              Waypoint Linea28_B: TCP in base x=-638.706 y=351.254 z=110.848 mm, rx=0.1163 ry=3.1217 rz=0.0052 rad; joints [-32.94, -74.396, 108.519, -33.495, -217.835, -0.377] deg
              Folder bajada_comprobacion
                MoveDirectionNode (selectedDirection=ZMinus toolParams=0.1, 0.15)
                  Until DISTANCE (allowActions=false deceleration=3 distanceNodeType=STOP) Distance=0.071; motionParameters(blendRadius=0)
                MoveDirectionNode (selectedDirection=ZMinus toolParams=0.007, 0.007)
                  Until TOOL_CONTACT_DETECTION (allowActions=false retraction=0 decelerationAcceleration=0.02 decelerationAngularAcceleration=34.906585)
                MoveDirectionNode (selectedDirection=ZPlus toolParams=0.1, 0.15)
                  Until DISTANCE (allowActions=false deceleration=3 distanceNodeType=STOP) Distance=0.08; motionParameters(blendRadius=0)
          Folder AB
            'desbaste_inicial'
            bajada_broca := p[0,0,-0.008,0,0,0]
            barrenos_menos1 := 0
            barreno_actual := 0
            Loop While (checkContinuously=false) expression=barreno_actual≤barrenos_menos1
              Folder Perforacion
                MoveL speed 100 mm/s, acceleration 500 mm/s^2 (useActiveTCP=true) feature=Base
                  SuppressedNode
                    If barreno_actual≟3
                      barreno_actual := barreno_actual+1
                  SuppressedNode
                    internos := interpolate_pose(Linea28_B, Linea28_B, barreno_actual/barrenos_menos1)
                  SuppressedNode
                    Waypoint Waypoint (Variable): variable=internos
                  Waypoint Linea28_B referenceName=Linea28_B: TCP in base x=-638.706 y=351.254 z=110.848 mm, rx=0.1163 ry=3.1217 rz=0.0052 rad; joints [-32.94, -74.396, 108.519, -33.495, -217.835, -0.377] deg
                  'desbaste_inicial'
                  bajada_broca := p[0,0,-0.024,0,0,0]
                  bajada := p[0,0,0.024,0,0,0]
                  MoveDirectionNode (selectedDirection=ZMinus toolParams=0.1, 0.15)
                    Until DISTANCE (allowActions=false deceleration=3 distanceNodeType=STOP) Distance=0.071; motionParameters(blendRadius=0)
                  MoveDirectionNode (selectedDirection=ZMinus toolParams=0.007, 0.007)
                    Until TOOL_CONTACT_DETECTION (allowActions=false retraction=0 decelerationAcceleration=0.02 decelerationAngularAcceleration=34.906585)
                  Popup Message (haltProgram=false message=punto contacto alanzdo inputType=Text)
                  MoveDirectionNode (selectedDirection=ZPlus toolParams=0.015, 0.015)
                    Until DISTANCE (allowActions=false deceleration=3 distanceNodeType=STOP) Distance=0.01; motionParameters(blendRadius=0)
                  Wait Sleep waitTime=0.3
                  Set DigitalOutput pin=config_out[1]; digitalValue=1
                  Wait Sleep waitTime=0.3
                  Loop Counting (count=1) loopVariable(name=Loop_146)
                    bajar := pose_add(get_actual_tcp_pose(), bajada_broca)
                    Waypoint Waypoint (Variable): motionParameters(jointSpeed=1.047198 jointAcceleration=1.396263 cartesianSpeed=0.004 cartesianAcceleration=0.004); variable=bajar
                    subir := pose_sub(get_actual_tcp_pose(), bajada_broca)
                    MoveDirectionNode (selectedDirection=ZPlus toolParams=0.015, 0.015)
                      Until DISTANCE (allowActions=false deceleration=3 distanceNodeType=STOP) Distance=0.002; motionParameters(blendRadius=0)
                    Set DigitalOutput pin=config_out[1]; digitalValue=0
                    Waypoint Waypoint (Variable): motionParameters(jointSpeed=1.047198 jointAcceleration=1.396263 cartesianSpeed=0.015 cartesianAcceleration=0.015); variable=subir
                    bajada_broca := pose_sub(bajada_broca, bajada)
                  MoveDirectionNode (selectedDirection=ZPlus toolParams=0.1, 0.15)
                    Until DISTANCE (allowActions=false deceleration=3 distanceNodeType=STOP) Distance=0.08; motionParameters(blendRadius=0)
                  Set DigitalOutput pin=config_out[1]; digitalValue=0
                  barreno_actual := barreno_actual+1
                  SuppressedNode
                    Call Quitar_broca
                  SuppressedNode
                    Call Poner_broca
        Popup Message (haltProgram=false message=Linea28 con chica Terminada! inputType=Text)
        Folder Linea29
          Folder Marcar_puntos
            MoveL speed 100 mm/s, acceleration 500 mm/s^2 (useActiveTCP=true) feature=Base
              Waypoint Linea29_A: TCP in base x=-697.642 y=-428.593 z=109.99 mm, rx=-2.8017 ry=1.4172 rz=0.0072 rad; joints [13.48, -73.278, 107.072, -33.144, -302.021, -0.481] deg; TCP offset x=0.411 y=-218.298 z=37.994 mm, rx=1.558 ry=-0.1255 rz=0.1212 rad
              SuppressedNode
                Waypoint Linea29_BA: TCP in base x=-927.927 y=-428.7 z=110.397 mm, rx=-2.8034 ry=1.4179 rz=0.011 rad; joints [9.956, -55.686, 80.201, -24.007, -305.531, -0.529] deg
              Folder bajada_comprobacion
                MoveDirectionNode (selectedDirection=ZMinus toolParams=0.1, 0.15)
                  Until DISTANCE (allowActions=false deceleration=3 distanceNodeType=STOP) Distance=0.071; motionParameters(blendRadius=0)
                MoveDirectionNode (selectedDirection=ZMinus toolParams=0.007, 0.007)
                  Until TOOL_CONTACT_DETECTION (allowActions=false retraction=0 decelerationAcceleration=0.02 decelerationAngularAcceleration=34.906585)
                MoveDirectionNode (selectedDirection=ZPlus toolParams=0.1, 0.15)
                  Until DISTANCE (allowActions=false deceleration=3 distanceNodeType=STOP) Distance=0.08; motionParameters(blendRadius=0)
              SuppressedNode
                Waypoint Linea29_B: TCP in base x=-1160.231 y=-428.651 z=110.797 mm, rx=-2.8017 ry=1.4172 rz=0.0072 rad; joints [7.841, -31.782, 37.108, -4.619, -307.592, -0.568] deg
              Waypoint Linea29_AB: TCP in base x=-904.922 y=-428.637 z=110.457 mm, rx=-2.8017 ry=1.4172 rz=0.0072 rad; joints [10.222, -57.489, 83.131, -24.963, -305.263, -0.527] deg
              Folder bajada_comprobacion
                MoveDirectionNode (selectedDirection=ZMinus toolParams=0.1, 0.15)
                  Until DISTANCE (allowActions=false deceleration=3 distanceNodeType=STOP) Distance=0.071; motionParameters(blendRadius=0)
                MoveDirectionNode (selectedDirection=ZMinus toolParams=0.007, 0.007)
                  Until TOOL_CONTACT_DETECTION (allowActions=false retraction=0 decelerationAcceleration=0.02 decelerationAngularAcceleration=34.906585)
                MoveDirectionNode (selectedDirection=ZPlus toolParams=0.1, 0.15)
                  Until DISTANCE (allowActions=false deceleration=3 distanceNodeType=STOP) Distance=0.08; motionParameters(blendRadius=0)
          Folder AB
            'desbaste_inicial'
            bajada_broca := p[0,0,-0.008,0,0,0]
            barrenos_menos1 := 9
            barreno_actual := 0
            Loop While (checkContinuously=false) expression=barreno_actual≤barrenos_menos1
              Folder Perforacion
                MoveL speed 100 mm/s, acceleration 500 mm/s^2 (useActiveTCP=true) feature=Base
                  If barreno_actual≟7
                    barreno_actual := barreno_actual+1
                  internos := interpolate_pose(Linea29_A, Linea29_AB, barreno_actual/barrenos_menos1)
                  SuppressedNode
                    If barreno_actual≟6
                      MoveDirectionNode (selectedDirection=ZPlus)
                        Until DISTANCE (allowActions=false deceleration=3 distanceNodeType=STOP) Distance=0.01; motionParameters(blendRadius=0)
                  Waypoint Waypoint (Variable): variable=internos
                  'desbaste_inicial'
                  bajada_broca := p[0,0,-0.024,0,0,0]
                  bajada := p[0,0,0.024,0,0,0]
                  MoveDirectionNode (selectedDirection=ZMinus toolParams=0.1, 0.15)
                    Until DISTANCE (allowActions=false deceleration=3 distanceNodeType=STOP) Distance=0.071; motionParameters(blendRadius=0)
                  MoveDirectionNode (selectedDirection=ZMinus toolParams=0.007, 0.007)
                    Until TOOL_CONTACT_DETECTION (allowActions=false retraction=0 decelerationAcceleration=0.02 decelerationAngularAcceleration=34.906585)
                  Popup Message (haltProgram=false message=punto contacto alanzdo inputType=Text)
                  MoveDirectionNode (selectedDirection=ZPlus toolParams=0.015, 0.015)
                    Until DISTANCE (allowActions=false deceleration=3 distanceNodeType=STOP) Distance=0.007; motionParameters(blendRadius=0)
                  Wait Sleep waitTime=0.3
                  Set DigitalOutput pin=config_out[1]; digitalValue=1
                  Wait Sleep waitTime=0.3
                  Loop Counting (count=1) loopVariable(name=Loop_150)
                    bajar := pose_add(get_actual_tcp_pose(), bajada_broca)
                    Waypoint Waypoint (Variable): motionParameters(jointSpeed=1.047198 jointAcceleration=1.396263 cartesianSpeed=0.004 cartesianAcceleration=0.004); variable=bajar
                    subir := pose_sub(get_actual_tcp_pose(), bajada_broca)
                    MoveDirectionNode (selectedDirection=ZPlus toolParams=0.015, 0.015)
                      Until DISTANCE (allowActions=false deceleration=3 distanceNodeType=STOP) Distance=0.002; motionParameters(blendRadius=0)
                    Set DigitalOutput pin=config_out[1]; digitalValue=0
                    Waypoint Waypoint (Variable): motionParameters(jointSpeed=1.047198 jointAcceleration=1.396263 cartesianSpeed=0.015 cartesianAcceleration=0.015); variable=subir
                    bajada_broca := pose_sub(bajada_broca, bajada)
                  MoveDirectionNode (selectedDirection=ZPlus toolParams=0.1, 0.15)
                    Until DISTANCE (allowActions=false deceleration=3 distanceNodeType=STOP) Distance=0.04; motionParameters(blendRadius=0)
                  Set DigitalOutput pin=config_out[1]; digitalValue=0
                  barreno_actual := barreno_actual+1
                  SuppressedNode
                    Call Quitar_broca
                  SuppressedNode
                    Call Poner_broca
        Folder Linea29B
          Folder Marcar_puntos
            MoveL speed 100 mm/s, acceleration 500 mm/s^2 (useActiveTCP=true) feature=Base
              SuppressedNode
                Waypoint Linea29_A: TCP in base x=-697.642 y=-428.593 z=109.99 mm, rx=-2.8017 ry=1.4172 rz=0.0072 rad; joints [13.48, -73.278, 107.072, -33.144, -302.021, -0.481] deg
              Waypoint Linea29_BA: TCP in base x=-927.927 y=-428.7 z=110.397 mm, rx=-2.8034 ry=1.4179 rz=0.011 rad; joints [9.956, -55.686, 80.201, -24.007, -305.531, -0.529] deg
              Folder bajada_comprobacion
                MoveDirectionNode (selectedDirection=ZMinus toolParams=0.1, 0.15)
                  Until DISTANCE (allowActions=false deceleration=3 distanceNodeType=STOP) Distance=0.071; motionParameters(blendRadius=0)
                MoveDirectionNode (selectedDirection=ZMinus toolParams=0.007, 0.007)
                  Until TOOL_CONTACT_DETECTION (allowActions=false retraction=0 decelerationAcceleration=0.02 decelerationAngularAcceleration=34.906585)
                MoveDirectionNode (selectedDirection=ZPlus toolParams=0.1, 0.15)
                  Until DISTANCE (allowActions=false deceleration=3 distanceNodeType=STOP) Distance=0.08; motionParameters(blendRadius=0)
              Waypoint Linea29_B: TCP in base x=-1160.231 y=-428.651 z=110.797 mm, rx=-2.8017 ry=1.4172 rz=0.0072 rad; joints [7.841, -31.782, 37.108, -4.619, -307.592, -0.568] deg
              SuppressedNode
                Waypoint Linea29_AB: TCP in base x=-904.922 y=-428.637 z=110.457 mm, rx=-2.8017 ry=1.4172 rz=0.0072 rad; joints [10.222, -57.489, 83.131, -24.963, -305.263, -0.527] deg
              Folder bajada_comprobacion
                MoveDirectionNode (selectedDirection=ZMinus toolParams=0.1, 0.15)
                  Until DISTANCE (allowActions=false deceleration=3 distanceNodeType=STOP) Distance=0.071; motionParameters(blendRadius=0)
                MoveDirectionNode (selectedDirection=ZMinus toolParams=0.007, 0.007)
                  Until TOOL_CONTACT_DETECTION (allowActions=false retraction=0 decelerationAcceleration=0.02 decelerationAngularAcceleration=34.906585)
                MoveDirectionNode (selectedDirection=ZPlus toolParams=0.1, 0.15)
                  Until DISTANCE (allowActions=false deceleration=3 distanceNodeType=STOP) Distance=0.08; motionParameters(blendRadius=0)
          Folder AB
            'desbaste_inicial'
            bajada_broca := p[0,0,-0.008,0,0,0]
            barrenos_menos1 := 10
            barreno_actual := 5
            Loop While (checkContinuously=false) expression=barreno_actual≤barrenos_menos1
              Folder Perforacion
                MoveL speed 100 mm/s, acceleration 500 mm/s^2 (useActiveTCP=true) feature=Base
                  SuppressedNode
                    If barreno_actual≟7
                      barreno_actual := barreno_actual+1
                  internos := interpolate_pose(Linea29_BA, Linea29_B, barreno_actual/barrenos_menos1)
                  SuppressedNode
                    If barreno_actual≟6
                      MoveDirectionNode (selectedDirection=ZPlus)
                        Until DISTANCE (allowActions=false deceleration=3 distanceNodeType=STOP) Distance=0.01; motionParameters(blendRadius=0)
                  Waypoint Waypoint (Variable): variable=internos
                  'desbaste_inicial'
                  bajada_broca := p[0,0,-0.024,0,0,0]
                  bajada := p[0,0,0.024,0,0,0]
                  MoveDirectionNode (selectedDirection=ZMinus toolParams=0.1, 0.15)
                    Until DISTANCE (allowActions=false deceleration=3 distanceNodeType=STOP) Distance=0.071; motionParameters(blendRadius=0)
                  MoveDirectionNode (selectedDirection=ZMinus toolParams=0.007, 0.007)
                    Until TOOL_CONTACT_DETECTION (allowActions=false retraction=0 decelerationAcceleration=0.02 decelerationAngularAcceleration=34.906585)
                  Popup Message (haltProgram=false message=punto contacto alanzdo inputType=Text)
                  MoveDirectionNode (selectedDirection=ZPlus toolParams=0.015, 0.015)
                    Until DISTANCE (allowActions=false deceleration=3 distanceNodeType=STOP) Distance=0.007; motionParameters(blendRadius=0)
                  Wait Sleep waitTime=0.3
                  Set DigitalOutput pin=config_out[1]; digitalValue=1
                  Wait Sleep waitTime=0.3
                  Loop Counting (count=1) loopVariable(name=Loop_30)
                    bajar := pose_add(get_actual_tcp_pose(), bajada_broca)
                    Waypoint Waypoint (Variable): motionParameters(jointSpeed=1.047198 jointAcceleration=1.396263 cartesianSpeed=0.004 cartesianAcceleration=0.004); variable=bajar
                    subir := pose_sub(get_actual_tcp_pose(), bajada_broca)
                    MoveDirectionNode (selectedDirection=ZPlus toolParams=0.015, 0.015)
                      Until DISTANCE (allowActions=false deceleration=3 distanceNodeType=STOP) Distance=0.002; motionParameters(blendRadius=0)
                    Set DigitalOutput pin=config_out[1]; digitalValue=0
                    Waypoint Waypoint (Variable): motionParameters(jointSpeed=1.047198 jointAcceleration=1.396263 cartesianSpeed=0.015 cartesianAcceleration=0.015); variable=subir
                    bajada_broca := pose_sub(bajada_broca, bajada)
                  MoveDirectionNode (selectedDirection=ZPlus toolParams=0.1, 0.15)
                    Until DISTANCE (allowActions=false deceleration=3 distanceNodeType=STOP) Distance=0.04; motionParameters(blendRadius=0)
                  Set DigitalOutput pin=config_out[1]; digitalValue=0
                  barreno_actual := barreno_actual+1
                  SuppressedNode
                    Call Quitar_broca
                  SuppressedNode
                    Call Poner_broca
        Popup Message (haltProgram=false message=Linea29 con chica Terminada! inputType=Text)
      SuppressedNode
        Folder Broca_2
          Folder Linea7
            Folder Marcar_puntos
              MoveL speed 100 mm/s, acceleration 500 mm/s^2 (useActiveTCP=true) feature=Base
                Waypoint Home2: TCP in base x=-476.229 y=0 z=568.737 mm, rx=2.0263 ry=-2.3929 rz=-0.0208 rad; joints [-32.551, -116.469, 98.413, 17.843, -302.102, -0.163] deg; TCP offset x=0.411 y=-218.298 z=37.994 mm, rx=1.558 ry=-0.1255 rz=0.1212 rad
                Waypoint Linea7_A: TCP in base x=-749.561 y=-351.839 z=110.843 mm, rx=3.1084 ry=-0.3759 rz=-0.0174 rad; joints [1.917, -65.95, 96.598, -30.808, -353.455, -0.309] deg
                Waypoint Linea7_B: TCP in base x=-795.37 y=-351.638 z=110.748 mm, rx=3.1084 ry=-0.3758 rz=-0.0174 rad; joints [1.792, -62.243, 90.906, -28.822, -353.578, -0.309] deg
            Folder AB
              'desbaste_inicial'
              bajada_broca := p[0,0,-0.008,0,0,0]
              barrenos_menos1 := 2
              barreno_actual := 0
              Loop While (checkContinuously=false) expression=barreno_actual≤barrenos_menos1
                Folder Perforacion
                  MoveL speed 100 mm/s, acceleration 500 mm/s^2 (useActiveTCP=true) feature=Base
                    internos := interpolate_pose(Linea7_A, Linea7_B, barreno_actual/barrenos_menos1)
                    Waypoint Waypoint (Variable): variable=internos
                    'desbaste_inicial'
                    bajada_broca := p[0,0,-0.008,0,0,0]
                    bajada := p[0,0,0.008,0,0,0]
                    MoveDirectionNode (selectedDirection=ZMinus toolParams=0.003, 0.005)
                      Until DISTANCE (allowActions=false deceleration=3 distanceNodeType=STOP) Distance=0.045; motionParameters(blendRadius=0)
                    Popup Message (haltProgram=false message=punto contacto alanzdo inputType=Text)
                    MoveDirectionNode (selectedDirection=ZPlus toolParams=0.003, 0.005)
                      Until DISTANCE (allowActions=false deceleration=3 distanceNodeType=STOP) Distance=0.002; motionParameters(blendRadius=0)
                    Wait Sleep waitTime=0.3
                    Set DigitalOutput pin=config_out[1]; digitalValue=1
                    Wait Sleep waitTime=0.3
                    Loop Counting (count=3) loopVariable(name=Loop_111)
                      bajar := pose_add(get_actual_tcp_pose(), bajada_broca)
                      Waypoint Waypoint (Variable): motionParameters(jointSpeed=1.047198 jointAcceleration=1.396263 cartesianSpeed=0.001 cartesianAcceleration=0.005); variable=bajar
                      subir := pose_sub(get_actual_tcp_pose(), bajada_broca)
                      Waypoint Waypoint (Variable): motionParameters(jointSpeed=1.047198 jointAcceleration=1.396263 cartesianSpeed=0.005 cartesianAcceleration=0.01); variable=subir
                      bajada_broca := pose_sub(bajada_broca, bajada)
                    MoveDirectionNode (selectedDirection=ZPlus toolParams=0.03, 0.035)
                      Until DISTANCE (allowActions=false deceleration=3 distanceNodeType=STOP) Distance=0.06; motionParameters(blendRadius=0)
                    Set DigitalOutput pin=config_out[1]; digitalValue=0
                    barreno_actual := barreno_actual+1
                    SuppressedNode
                      Call Quitar_broca
                    SuppressedNode
                      Call Poner_broca
          Popup Message (haltProgram=false message=Linea7 con chica Terminada! inputType=Text)
          Folder Linea8
            Folder Marcar_puntos
              MoveL speed 100 mm/s, acceleration 500 mm/s^2 (useActiveTCP=true) feature=Base
                Waypoint Linea8_A: TCP in base x=-897.665 y=-351.421 z=100.251 mm, rx=3.1084 ry=-0.3758 rz=-0.0174 rad; joints [1.574, -53.233, 77.321, -24.256, -353.784, -0.302] deg
                Waypoint Linea8_B: TCP in base x=-1021.743 y=-350.913 z=110.77 mm, rx=3.1084 ry=-0.3758 rz=-0.0173 rad; joints [1.351, -41.656, 55.75, -14.225, -353.984, -0.335] deg
            Folder AB
              'desbaste_inicial'
              bajada_broca := p[0,0,-0.008,0,0,0]
              barrenos_menos1 := 5
              barreno_actual := 0
              Loop While (checkContinuously=false) expression=barreno_actual≤barrenos_menos1
                Folder Perforacion
                  MoveL speed 100 mm/s, acceleration 500 mm/s^2 (useActiveTCP=true) feature=Base
                    internos := interpolate_pose(Linea8_A, Linea8_B, barreno_actual/barrenos_menos1)
                    Waypoint Waypoint (Variable): variable=internos
                    'desbaste_inicial'
                    bajada_broca := p[0,0,-0.008,0,0,0]
                    bajada := p[0,0,0.008,0,0,0]
                    MoveDirectionNode (selectedDirection=ZMinus toolParams=0.003, 0.005)
                      Until DISTANCE (allowActions=false deceleration=3 distanceNodeType=STOP) Distance=0.045; motionParameters(blendRadius=0)
                    Popup Message (haltProgram=false message=punto contacto alanzdo inputType=Text)
                    MoveDirectionNode (selectedDirection=ZPlus toolParams=0.003, 0.005)
                      Until DISTANCE (allowActions=false deceleration=3 distanceNodeType=STOP) Distance=0.002; motionParameters(blendRadius=0)
                    Wait Sleep waitTime=0.3
                    Set DigitalOutput pin=config_out[1]; digitalValue=1
                    Wait Sleep waitTime=0.3
                    Loop Counting (count=3) loopVariable(name=Loop_113)
                      bajar := pose_add(get_actual_tcp_pose(), bajada_broca)
                      Waypoint Waypoint (Variable): motionParameters(jointSpeed=1.047198 jointAcceleration=1.396263 cartesianSpeed=0.001 cartesianAcceleration=0.005); variable=bajar
                      subir := pose_sub(get_actual_tcp_pose(), bajada_broca)
                      Waypoint Waypoint (Variable): motionParameters(jointSpeed=1.047198 jointAcceleration=1.396263 cartesianSpeed=0.005 cartesianAcceleration=0.01); variable=subir
                      bajada_broca := pose_sub(bajada_broca, bajada)
                    MoveDirectionNode (selectedDirection=ZPlus toolParams=0.03, 0.035)
                      Until DISTANCE (allowActions=false deceleration=3 distanceNodeType=STOP) Distance=0.06; motionParameters(blendRadius=0)
                    Set DigitalOutput pin=config_out[1]; digitalValue=0
                    barreno_actual := barreno_actual+1
                    SuppressedNode
                      Call Quitar_broca
                    SuppressedNode
                      Call Poner_broca
          Popup Message (haltProgram=false message=Linea8 con chica Terminada! inputType=Text)
          Folder Linea9
            Folder Marcar_puntos
              MoveL speed 100 mm/s, acceleration 500 mm/s^2 (useActiveTCP=true) feature=Base
                Waypoint Linea9_A: TCP in base x=-1101.087 y=-350.536 z=110.686 mm, rx=3.1084 ry=-0.3759 rz=-0.0174 rad; joints [1.23, -31.558, 36.849, -5.411, -354.078, -0.351] deg
                Waypoint Linea9_B: TCP in base x=-1151 y=-350.505 z=110.708 mm, rx=3.1084 ry=-0.3759 rz=-0.0174 rad; joints [1.169, -21.153, 16.449, 4.577, -354.109, -0.341] deg
            Folder AB
              'desbaste_inicial'
              bajada_broca := p[0,0,-0.008,0,0,0]
              barrenos_menos1 := 2
              barreno_actual := 0
              Loop While (checkContinuously=false) expression=barreno_actual≤barrenos_menos1
                Folder Perforacion
                  MoveL speed 100 mm/s, acceleration 500 mm/s^2 (useActiveTCP=true) feature=Base
                    internos := interpolate_pose(Linea9_A, Linea9_B, barreno_actual/barrenos_menos1)
                    Waypoint Waypoint (Variable): variable=internos
                    'desbaste_inicial'
                    bajada_broca := p[0,0,-0.008,0,0,0]
                    bajada := p[0,0,0.008,0,0,0]
                    MoveDirectionNode (selectedDirection=ZMinus toolParams=0.003, 0.005)
                      Until DISTANCE (allowActions=false deceleration=3 distanceNodeType=STOP) Distance=0.045; motionParameters(blendRadius=0)
                    Popup Message (haltProgram=false message=punto contacto alanzdo inputType=Text)
                    MoveDirectionNode (selectedDirection=ZPlus toolParams=0.003, 0.005)
                      Until DISTANCE (allowActions=false deceleration=3 distanceNodeType=STOP) Distance=0.002; motionParameters(blendRadius=0)
                    Wait Sleep waitTime=0.3
                    Set DigitalOutput pin=config_out[1]; digitalValue=1
                    Wait Sleep waitTime=0.3
                    Loop Counting (count=3) loopVariable(name=Loop_115)
                      bajar := pose_add(get_actual_tcp_pose(), bajada_broca)
                      Waypoint Waypoint (Variable): motionParameters(jointSpeed=1.047198 jointAcceleration=1.396263 cartesianSpeed=0.001 cartesianAcceleration=0.005); variable=bajar
                      subir := pose_sub(get_actual_tcp_pose(), bajada_broca)
                      Waypoint Waypoint (Variable): motionParameters(jointSpeed=1.047198 jointAcceleration=1.396263 cartesianSpeed=0.005 cartesianAcceleration=0.01); variable=subir
                      bajada_broca := pose_sub(bajada_broca, bajada)
                    MoveDirectionNode (selectedDirection=ZPlus toolParams=0.03, 0.035)
                      Until DISTANCE (allowActions=false deceleration=3 distanceNodeType=STOP) Distance=0.06; motionParameters(blendRadius=0)
                    Set DigitalOutput pin=config_out[1]; digitalValue=0
                    barreno_actual := barreno_actual+1
                    SuppressedNode
                      Call Quitar_broca
                    SuppressedNode
                      Call Poner_broca
          Popup Message (haltProgram=false message=Linea9 con chica Terminada! inputType=Text)
          Folder Linea10
            Folder Marcar_puntos
              MoveL speed 100 mm/s, acceleration 500 mm/s^2 (useActiveTCP=true) feature=Base
                Waypoint Home2: TCP in base x=-476.229 y=0 z=568.737 mm, rx=2.0263 ry=-2.3929 rz=-0.0208 rad; joints [-32.551, -116.469, 98.413, 17.843, -302.102, -0.163] deg
                Waypoint Linea10_A: TCP in base x=-634.372 y=-317.237 z=110 mm, rx=3.1084 ry=-0.3759 rz=-0.0173 rad; joints [-0.923, -75.994, 110.915, -35.183, -356.299, -0.201] deg
                Waypoint Linea10_B: TCP in base x=-637.528 y=-266.765 z=110 mm, rx=2.0205 ry=-2.3939 rz=-0.0206 rad; joints [10.666, -83.833, 120.67, -37.235, -258.835, -0.176] deg
            Folder AB
              'desbaste_inicial'
              bajada_broca := p[0,0,-0.008,0,0,0]
              barrenos_menos1 := 2
              barreno_actual := 0
              Loop While (checkContinuously=false) expression=barreno_actual≤barrenos_menos1
                Folder Perforacion
                  MoveL speed 100 mm/s, acceleration 500 mm/s^2 (useActiveTCP=true) feature=Base
                    internos := interpolate_pose(Linea10_A, Linea10_B, barreno_actual/barrenos_menos1)
                    Waypoint Waypoint (Variable): variable=internos
                    'desbaste_inicial'
                    bajada_broca := p[0,0,-0.008,0,0,0]
                    bajada := p[0,0,0.008,0,0,0]
                    MoveDirectionNode (selectedDirection=ZMinus toolParams=0.003, 0.005)
                      Until DISTANCE (allowActions=false deceleration=3 distanceNodeType=STOP) Distance=0.045; motionParameters(blendRadius=0)
                    Popup Message (haltProgram=false message=punto contacto alanzdo inputType=Text)
                    MoveDirectionNode (selectedDirection=ZPlus toolParams=0.003, 0.005)
                      Until DISTANCE (allowActions=false deceleration=3 distanceNodeType=STOP) Distance=0.002; motionParameters(blendRadius=0)
                    Wait Sleep waitTime=0.3
                    Set DigitalOutput pin=config_out[1]; digitalValue=1
                    Wait Sleep waitTime=0.3
                    Loop Counting (count=3) loopVariable(name=Loop_117)
                      bajar := pose_add(get_actual_tcp_pose(), bajada_broca)
                      Waypoint Waypoint (Variable): motionParameters(jointSpeed=1.047198 jointAcceleration=1.396263 cartesianSpeed=0.001 cartesianAcceleration=0.005); variable=bajar
                      subir := pose_sub(get_actual_tcp_pose(), bajada_broca)
                      Waypoint Waypoint (Variable): motionParameters(jointSpeed=1.047198 jointAcceleration=1.396263 cartesianSpeed=0.005 cartesianAcceleration=0.01); variable=subir
                      bajada_broca := pose_sub(bajada_broca, bajada)
                    MoveDirectionNode (selectedDirection=ZPlus toolParams=0.03, 0.035)
                      Until DISTANCE (allowActions=false deceleration=3 distanceNodeType=STOP) Distance=0.06; motionParameters(blendRadius=0)
                    Set DigitalOutput pin=config_out[1]; digitalValue=0
                    barreno_actual := barreno_actual+1
                    SuppressedNode
                      Call Quitar_broca
                    SuppressedNode
                      Call Poner_broca
          Popup Message (haltProgram=false message=Linea10 con chica Terminada! inputType=Text)
          Folder Linea11
            Folder Marcar_puntos
              MoveL speed 100 mm/s, acceleration 500 mm/s^2 (useActiveTCP=true) feature=Base
                Waypoint Linea11_A: TCP in base x=-636.9 y=-137.433 z=110 mm, rx=2.0204 ry=-2.394 rz=-0.0205 rad; joints [-4.253, -88.617, 125.878, -37.636, -273.75, -0.078] deg
                Waypoint Linea11_B: TCP in base x=-636.767 y=-82.891 z=110 mm, rx=2.0204 ry=-2.3939 rz=-0.0206 rad; joints [-10.939, -89.848, 127.132, -37.66, -280.436, -0.033] deg
            Folder AB
              'desbaste_inicial'
              bajada_broca := p[0,0,-0.008,0,0,0]
              barrenos_menos1 := 2
              barreno_actual := 0
              Loop While (checkContinuously=false) expression=barreno_actual≤barrenos_menos1
                Folder Perforacion
                  MoveL speed 100 mm/s, acceleration 500 mm/s^2 (useActiveTCP=true) feature=Base
                    SuppressedNode
                      If barreno_actual≟5
                        barreno_actual := barreno_actual+1
                    internos := interpolate_pose(Linea11_A, Linea11_B, barreno_actual/barrenos_menos1)
                    Waypoint Waypoint (Variable): variable=internos
                    'desbaste_inicial'
                    bajada_broca := p[0,0,-0.008,0,0,0]
                    bajada := p[0,0,0.008,0,0,0]
                    MoveDirectionNode (selectedDirection=ZMinus toolParams=0.003, 0.005)
                      Until DISTANCE (allowActions=false deceleration=3 distanceNodeType=STOP) Distance=0.045; motionParameters(blendRadius=0)
                    Popup Message (haltProgram=false message=punto contacto alanzdo inputType=Text)
                    MoveDirectionNode (selectedDirection=ZPlus toolParams=0.003, 0.005)
                      Until DISTANCE (allowActions=false deceleration=3 distanceNodeType=STOP) Distance=0.002; motionParameters(blendRadius=0)
                    Wait Sleep waitTime=0.3
                    Set DigitalOutput pin=config_out[1]; digitalValue=1
                    Wait Sleep waitTime=0.3
                    Loop Counting (count=3) loopVariable(name=Loop_119)
                      bajar := pose_add(get_actual_tcp_pose(), bajada_broca)
                      Waypoint Waypoint (Variable): motionParameters(jointSpeed=1.047198 jointAcceleration=1.396263 cartesianSpeed=0.001 cartesianAcceleration=0.005); variable=bajar
                      subir := pose_sub(get_actual_tcp_pose(), bajada_broca)
                      Waypoint Waypoint (Variable): motionParameters(jointSpeed=1.047198 jointAcceleration=1.396263 cartesianSpeed=0.005 cartesianAcceleration=0.01); variable=subir
                      bajada_broca := pose_sub(bajada_broca, bajada)
                    MoveDirectionNode (selectedDirection=ZPlus toolParams=0.03, 0.035)
                      Until DISTANCE (allowActions=false deceleration=3 distanceNodeType=STOP) Distance=0.06; motionParameters(blendRadius=0)
                    Set DigitalOutput pin=config_out[1]; digitalValue=0
                    barreno_actual := barreno_actual+1
                    SuppressedNode
                      Call Quitar_broca
                    SuppressedNode
                      Call Poner_broca
          Popup Message (haltProgram=false message=Linea11 con chica Terminada! inputType=Text)
          Folder Linea12
            Folder Marcar_puntos
              MoveL speed 100 mm/s, acceleration 500 mm/s^2 (useActiveTCP=true) feature=Base
                Waypoint Linea12_A: TCP in base x=-636.731 y=-59.028 z=110 mm, rx=2.0204 ry=-2.3939 rz=-0.0205 rad; joints [-13.873, -90.206, 127.489, -37.657, -283.371, -0.016] deg
                Waypoint Linea12_B: TCP in base x=-636.063 y=114.709 z=110 mm, rx=2.0204 ry=-2.3939 rz=-0.0206 rad; joints [-33.88, -89.351, 126.631, -37.694, -303.38, 0.135] deg
            Folder AB
              'desbaste_inicial'
              bajada_broca := p[0,0,-0.008,0,0,0]
              barrenos_menos1 := 7
              barreno_actual := 0
              Loop While (checkContinuously=false) expression=barreno_actual≤barrenos_menos1
                Folder Perforacion
                  MoveL speed 100 mm/s, acceleration 500 mm/s^2 (useActiveTCP=true) feature=Base
                    If barreno_actual≟2
                      barreno_actual := barreno_actual+1
                    internos := interpolate_pose(Linea12_A, Linea12_B, barreno_actual/barrenos_menos1)
                    Waypoint Waypoint (Variable): variable=internos
                    'desbaste_inicial'
                    bajada_broca := p[0,0,-0.008,0,0,0]
                    bajada := p[0,0,0.008,0,0,0]
                    MoveDirectionNode (selectedDirection=ZMinus toolParams=0.003, 0.005)
                      Until DISTANCE (allowActions=false deceleration=3 distanceNodeType=STOP) Distance=0.045; motionParameters(blendRadius=0)
                    Popup Message (haltProgram=false message=punto contacto alanzdo inputType=Text)
                    MoveDirectionNode (selectedDirection=ZPlus toolParams=0.003, 0.005)
                      Until DISTANCE (allowActions=false deceleration=3 distanceNodeType=STOP) Distance=0.002; motionParameters(blendRadius=0)
                    Wait Sleep waitTime=0.3
                    Set DigitalOutput pin=config_out[1]; digitalValue=1
                    Wait Sleep waitTime=0.3
                    Loop Counting (count=3) loopVariable(name=Loop_121)
                      bajar := pose_add(get_actual_tcp_pose(), bajada_broca)
                      Waypoint Waypoint (Variable): motionParameters(jointSpeed=1.047198 jointAcceleration=1.396263 cartesianSpeed=0.001 cartesianAcceleration=0.005); variable=bajar
                      subir := pose_sub(get_actual_tcp_pose(), bajada_broca)
                      Waypoint Waypoint (Variable): motionParameters(jointSpeed=1.047198 jointAcceleration=1.396263 cartesianSpeed=0.005 cartesianAcceleration=0.01); variable=subir
                      bajada_broca := pose_sub(bajada_broca, bajada)
                    MoveDirectionNode (selectedDirection=ZPlus toolParams=0.03, 0.035)
                      Until DISTANCE (allowActions=false deceleration=3 distanceNodeType=STOP) Distance=0.06; motionParameters(blendRadius=0)
                    Set DigitalOutput pin=config_out[1]; digitalValue=0
                    barreno_actual := barreno_actual+1
                    SuppressedNode
                      Call Quitar_broca
                    SuppressedNode
                      Call Poner_broca
          Popup Message (haltProgram=false message=Linea12 con chica Terminada! inputType=Text)
          Folder Linea13
            Folder Marcar_puntos
              MoveL speed 100 mm/s, acceleration 500 mm/s^2 (useActiveTCP=true) feature=Base
                Waypoint Linea13_A: TCP in base x=-636.036 y=270.318 z=110 mm, rx=2.0205 ry=-2.3939 rz=-0.0206 rad; joints [-47.614, -83.952, 120.807, -37.347, -317.114, 0.279] deg
                Waypoint Linea13_B: TCP in base x=-635.536 y=326.664 z=110 mm, rx=2.0205 ry=-2.3939 rz=-0.0206 rad; joints [-51.543, -81.32, 117.724, -36.932, -321.042, 0.336] deg
            Folder AB
              'desbaste_inicial'
              bajada_broca := p[0,0,-0.008,0,0,0]
              barrenos_menos1 := 2
              barreno_actual := 0
              Loop While (checkContinuously=false) expression=barreno_actual≤barrenos_menos1
                Folder Perforacion
                  MoveL speed 100 mm/s, acceleration 500 mm/s^2 (useActiveTCP=true) feature=Base
                    SuppressedNode
                      If barreno_actual≟2
                        barreno_actual := barreno_actual+1
                    internos := interpolate_pose(Linea13_A, Linea13_B, barreno_actual/barrenos_menos1)
                    Waypoint Waypoint (Variable): variable=internos
                    'desbaste_inicial'
                    bajada_broca := p[0,0,-0.008,0,0,0]
                    bajada := p[0,0,0.008,0,0,0]
                    MoveDirectionNode (selectedDirection=ZMinus toolParams=0.003, 0.005)
                      Until DISTANCE (allowActions=false deceleration=3 distanceNodeType=STOP) Distance=0.045; motionParameters(blendRadius=0)
                    Popup Message (haltProgram=false message=punto contacto alanzdo inputType=Text)
                    MoveDirectionNode (selectedDirection=ZPlus toolParams=0.003, 0.005)
                      Until DISTANCE (allowActions=false deceleration=3 distanceNodeType=STOP) Distance=0.002; motionParameters(blendRadius=0)
                    Wait Sleep waitTime=0.3
                    Set DigitalOutput pin=config_out[1]; digitalValue=1
                    Wait Sleep waitTime=0.3
                    Loop Counting (count=3) loopVariable=Loop_123
                      bajar := pose_add(get_actual_tcp_pose(), bajada_broca)
                      Waypoint Waypoint (Variable): motionParameters(jointSpeed=1.047198 jointAcceleration=1.396263 cartesianSpeed=0.001 cartesianAcceleration=0.005); variable=bajar
                      subir := pose_sub(get_actual_tcp_pose(), bajada_broca)
                      Waypoint Waypoint (Variable): motionParameters(jointSpeed=1.047198 jointAcceleration=1.396263 cartesianSpeed=0.005 cartesianAcceleration=0.01); variable=subir
                      bajada_broca := pose_sub(bajada_broca, bajada)
                    MoveDirectionNode (selectedDirection=ZPlus toolParams=0.03, 0.035)
                      Until DISTANCE (allowActions=false deceleration=3 distanceNodeType=STOP) Distance=0.06; motionParameters(blendRadius=0)
                    Set DigitalOutput pin=config_out[1]; digitalValue=0
                    barreno_actual := barreno_actual+1
                    SuppressedNode
                      Call Quitar_broca
                    SuppressedNode
                      Call Poner_broca
          Popup Message (haltProgram=false message=Linea13 con chica Terminada! inputType=Text)
          Folder Linea14
            Folder Marcar_puntos
              MoveL speed 100 mm/s, acceleration 500 mm/s^2 (useActiveTCP=true) feature=Base
                Waypoint Linea14_A: TCP in base x=-635.47 y=349.602 z=110 mm, rx=2.0205 ry=-2.3938 rz=-0.0205 rad; joints [-52.983, -80.161, 116.316, -36.699, -322.484, 0.362] deg
                Waypoint Linea14_B: TCP in base x=-634.908 y=491.921 z=110 mm, rx=2.0205 ry=-2.3939 rz=-0.0205 rad; joints [-60.308, -72.235, 105.919, -34.338, -329.805, 0.501] deg
            Folder AB
              'desbaste_inicial'
              bajada_broca := p[0,0,-0.008,0,0,0]
              barrenos_menos1 := 5
              barreno_actual := 0
              Loop While (checkContinuously=false) expression=barreno_actual≤barrenos_menos1
                Folder Perforacion
                  MoveL speed 100 mm/s, acceleration 500 mm/s^2 (useActiveTCP=true) feature=Base
                    If barreno_actual≟3
                      barreno_actual := barreno_actual+1
                    internos := interpolate_pose(Linea14_A, Linea14_B, barreno_actual/barrenos_menos1)
                    Waypoint Waypoint (Variable): variable=internos
                    'desbaste_inicial'
                    bajada_broca := p[0,0,-0.008,0,0,0]
                    bajada := p[0,0,0.008,0,0,0]
                    MoveDirectionNode (selectedDirection=ZMinus toolParams=0.003, 0.005)
                      Until DISTANCE (allowActions=false deceleration=3 distanceNodeType=STOP) Distance=0.045; motionParameters(blendRadius=0)
                    Popup Message (haltProgram=false message=punto contacto alanzdo inputType=Text)
                    MoveDirectionNode (selectedDirection=ZPlus toolParams=0.003, 0.005)
                      Until DISTANCE (allowActions=false deceleration=3 distanceNodeType=STOP) Distance=0.002; motionParameters(blendRadius=0)
                    Wait Sleep waitTime=0.3
                    Set DigitalOutput pin=config_out[1]; digitalValue=1
                    Wait Sleep waitTime=0.3
                    Loop Counting (count=3) loopVariable=Loop_125
                      bajar := pose_add(get_actual_tcp_pose(), bajada_broca)
                      Waypoint Waypoint (Variable): motionParameters(jointSpeed=1.047198 jointAcceleration=1.396263 cartesianSpeed=0.001 cartesianAcceleration=0.005); variable=bajar
                      subir := pose_sub(get_actual_tcp_pose(), bajada_broca)
                      Waypoint Waypoint (Variable): motionParameters(jointSpeed=1.047198 jointAcceleration=1.396263 cartesianSpeed=0.005 cartesianAcceleration=0.01); variable=subir
                      bajada_broca := pose_sub(bajada_broca, bajada)
                    MoveDirectionNode (selectedDirection=ZPlus toolParams=0.03, 0.035)
                      Until DISTANCE (allowActions=false deceleration=3 distanceNodeType=STOP) Distance=0.06; motionParameters(blendRadius=0)
                    Set DigitalOutput pin=config_out[1]; digitalValue=0
                    barreno_actual := barreno_actual+1
                    SuppressedNode
                      Call Quitar_broca
                    SuppressedNode
                      Call Poner_broca
          Popup Message (haltProgram=false message=Linea14 con chica Terminada! inputType=Text)
          Folder Linea15
            Folder Marcar_puntos
              MoveL speed 100 mm/s, acceleration 500 mm/s^2 (useActiveTCP=true) feature=Base
                Waypoint Linea15_A: TCP in base x=-634.597 y=515.429 z=110 mm, rx=2.0204 ry=-2.394 rz=-0.0205 rad; joints [-61.306, -70.837, 103.953, -33.788, -330.797, 0.523] deg
                Waypoint Linea15_B: TCP in base x=-634.619 y=593.839 z=110 mm, rx=2.0204 ry=-2.3939 rz=-0.0206 rad; joints [-64.194, -65.927, 96.758, -31.573, -333.685, 0.603] deg
            Folder AB
              'desbaste_inicial'
              bajada_broca := p[0,0,-0.008,0,0,0]
              barrenos_menos1 := 3
              barreno_actual := 0
              Loop While (checkContinuously=false) expression=barreno_actual≤barrenos_menos1
                Folder Perforacion
                  MoveL speed 100 mm/s, acceleration 500 mm/s^2 (useActiveTCP=true) feature=Base
                    SuppressedNode
                      If barreno_actual≟3
                        barreno_actual := barreno_actual+1
                    internos := interpolate_pose(Linea15_A, Linea15_B, barreno_actual/barrenos_menos1)
                    Waypoint Waypoint (Variable): variable=internos
                    'desbaste_inicial'
                    bajada_broca := p[0,0,-0.008,0,0,0]
                    bajada := p[0,0,0.008,0,0,0]
                    MoveDirectionNode (selectedDirection=ZMinus toolParams=0.003, 0.005)
                      Until DISTANCE (allowActions=false deceleration=3 distanceNodeType=STOP) Distance=0.045; motionParameters(blendRadius=0)
                    Popup Message (haltProgram=false message=punto contacto alanzdo inputType=Text)
                    MoveDirectionNode (selectedDirection=ZPlus toolParams=0.003, 0.005)
                      Until DISTANCE (allowActions=false deceleration=3 distanceNodeType=STOP) Distance=0.002; motionParameters(blendRadius=0)
                    Wait Sleep waitTime=0.3
                    Set DigitalOutput pin=config_out[1]; digitalValue=1
                    Wait Sleep waitTime=0.3
                    Loop Counting (count=3) loopVariable=Loop_127
                      bajar := pose_add(get_actual_tcp_pose(), bajada_broca)
                      Waypoint Waypoint (Variable): motionParameters(jointSpeed=1.047198 jointAcceleration=1.396263 cartesianSpeed=0.001 cartesianAcceleration=0.005); variable=bajar
                      subir := pose_sub(get_actual_tcp_pose(), bajada_broca)
                      Waypoint Waypoint (Variable): motionParameters(jointSpeed=1.047198 jointAcceleration=1.396263 cartesianSpeed=0.005 cartesianAcceleration=0.01); variable=subir
                      bajada_broca := pose_sub(bajada_broca, bajada)
                    MoveDirectionNode (selectedDirection=ZPlus toolParams=0.03, 0.035)
                      Until DISTANCE (allowActions=false deceleration=3 distanceNodeType=STOP) Distance=0.06; motionParameters(blendRadius=0)
                    Set DigitalOutput pin=config_out[1]; digitalValue=0
                    barreno_actual := barreno_actual+1
                    SuppressedNode
                      Call Quitar_broca
                    SuppressedNode
                      Call Poner_broca
          Popup Message (haltProgram=false message=Linea15 con chica Terminada! inputType=Text)
          Folder Linea16
            Folder Marcar_puntos
              MoveL speed 100 mm/s, acceleration 500 mm/s^2 (useActiveTCP=true) feature=Base
                Waypoint Linea16_A: TCP in base x=-471.483 y=617.988 z=110 mm, rx=-0.2145 ry=-3.1278 rz=-0.004 rad; joints [-60.34, -74.471, 108.758, -33.954, -241.667, 0.659] deg
                Waypoint Linea16_B: TCP in base x=-495.125 y=617.963 z=110 mm, rx=-0.2145 ry=-3.1278 rz=-0.004 rad; joints [-58.527, -73.043, 106.812, -33.43, -239.851, 0.673] deg
            Folder AB
              'desbaste_inicial'
              bajada_broca := p[0,0,-0.008,0,0,0]
              barrenos_menos1 := 1
              barreno_actual := 0
              Loop While (checkContinuously=false) expression=barreno_actual≤barrenos_menos1
                Folder Perforacion
                  MoveL speed 100 mm/s, acceleration 500 mm/s^2 (useActiveTCP=true) feature=Base
                    SuppressedNode
                      If barreno_actual≟3
                        barreno_actual := barreno_actual+1
                    internos := interpolate_pose(Linea16_A, Linea16_B, barreno_actual/barrenos_menos1)
                    Waypoint Waypoint (Variable): variable=internos
                    'desbaste_inicial'
                    bajada_broca := p[0,0,-0.008,0,0,0]
                    bajada := p[0,0,0.008,0,0,0]
                    MoveDirectionNode (selectedDirection=ZMinus toolParams=0.003, 0.005)
                      Until DISTANCE (allowActions=false deceleration=3 distanceNodeType=STOP) Distance=0.045; motionParameters(blendRadius=0)
                    Popup Message (haltProgram=false message=punto contacto alanzdo inputType=Text)
                    MoveDirectionNode (selectedDirection=ZPlus toolParams=0.003, 0.005)
                      Until DISTANCE (allowActions=false deceleration=3 distanceNodeType=STOP) Distance=0.002; motionParameters(blendRadius=0)
                    Wait Sleep waitTime=0.3
                    Set DigitalOutput pin=config_out[1]; digitalValue=1
                    Wait Sleep waitTime=0.3
                    Loop Counting (count=3) loopVariable=Loop_129
                      bajar := pose_add(get_actual_tcp_pose(), bajada_broca)
                      Waypoint Waypoint (Variable): motionParameters(jointSpeed=1.047198 jointAcceleration=1.396263 cartesianSpeed=0.001 cartesianAcceleration=0.005); variable=bajar
                      subir := pose_sub(get_actual_tcp_pose(), bajada_broca)
                      Waypoint Waypoint (Variable): motionParameters(jointSpeed=1.047198 jointAcceleration=1.396263 cartesianSpeed=0.005 cartesianAcceleration=0.01); variable=subir
                      bajada_broca := pose_sub(bajada_broca, bajada)
                    MoveDirectionNode (selectedDirection=ZPlus toolParams=0.03, 0.035)
                      Until DISTANCE (allowActions=false deceleration=3 distanceNodeType=STOP) Distance=0.06; motionParameters(blendRadius=0)
                    Set DigitalOutput pin=config_out[1]; digitalValue=0
                    barreno_actual := barreno_actual+1
                    SuppressedNode
                      Call Quitar_broca
                    SuppressedNode
                      Call Poner_broca
          Popup Message (haltProgram=false message=Linea16 con chica Terminada! inputType=Text)
          Folder Linea17
            Folder Marcar_puntos
              MoveL speed 100 mm/s, acceleration 500 mm/s^2 (useActiveTCP=true) feature=Base
                Waypoint Linea17_A: TCP in base x=-524.036 y=618.141 z=110 mm, rx=-0.2145 ry=-3.1278 rz=-0.0039 rad; joints [-56.431, -71.251, 104.315, -32.716, -237.756, 0.687] deg
                Waypoint Linea17_B: TCP in base x=-575.15 y=618.661 z=110 mm, rx=-0.2145 ry=-3.1278 rz=-0.0039 rad; joints [-53.015, -67.988, 99.609, -31.264, -234.337, 0.713] deg
            Folder AB
              'desbaste_inicial'
              bajada_broca := p[0,0,-0.008,0,0,0]
              barrenos_menos1 := 2
              barreno_actual := 0
              Loop While (checkContinuously=false) expression=barreno_actual≤barrenos_menos1
                Folder Perforacion
                  MoveL speed 100 mm/s, acceleration 500 mm/s^2 (useActiveTCP=true) feature=Base
                    SuppressedNode
                      If barreno_actual≟3
                        barreno_actual := barreno_actual+1
                    internos := interpolate_pose(Linea17_A, Linea17_B, barreno_actual/barrenos_menos1)
                    Waypoint Waypoint (Variable): variable=internos
                    'desbaste_inicial'
                    bajada_broca := p[0,0,-0.008,0,0,0]
                    bajada := p[0,0,0.008,0,0,0]
                    MoveDirectionNode (selectedDirection=ZMinus toolParams=0.003, 0.005)
                      Until DISTANCE (allowActions=false deceleration=3 distanceNodeType=STOP) Distance=0.045; motionParameters(blendRadius=0)
                    Popup Message (haltProgram=false message=punto contacto alanzdo inputType=Text)
                    MoveDirectionNode (selectedDirection=ZPlus toolParams=0.003, 0.005)
                      Until DISTANCE (allowActions=false deceleration=3 distanceNodeType=STOP) Distance=0.002; motionParameters(blendRadius=0)
                    Wait Sleep waitTime=0.3
                    Set DigitalOutput pin=config_out[1]; digitalValue=1
                    Wait Sleep waitTime=0.3
                    Loop Counting (count=3) loopVariable=Loop_131
                      bajar := pose_add(get_actual_tcp_pose(), bajada_broca)
                      Waypoint Waypoint (Variable): motionParameters(jointSpeed=1.047198 jointAcceleration=1.396263 cartesianSpeed=0.001 cartesianAcceleration=0.005); variable=bajar
                      subir := pose_sub(get_actual_tcp_pose(), bajada_broca)
                      Waypoint Waypoint (Variable): motionParameters(jointSpeed=1.047198 jointAcceleration=1.396263 cartesianSpeed=0.005 cartesianAcceleration=0.01); variable=subir
                      bajada_broca := pose_sub(bajada_broca, bajada)
                    MoveDirectionNode (selectedDirection=ZPlus toolParams=0.03, 0.035)
                      Until DISTANCE (allowActions=false deceleration=3 distanceNodeType=STOP) Distance=0.06; motionParameters(blendRadius=0)
                    Set DigitalOutput pin=config_out[1]; digitalValue=0
                    barreno_actual := barreno_actual+1
                    SuppressedNode
                      Call Quitar_broca
                    SuppressedNode
                      Call Poner_broca
          Popup Message (haltProgram=false message=Linea17 con chica Terminada! inputType=Text)
          Folder Linea18
            Folder Marcar_puntos
              MoveL speed 100 mm/s, acceleration 500 mm/s^2 (useActiveTCP=true) feature=Base
                Waypoint Linea18_A: TCP in base x=-659.545 y=625.386 z=80.084 mm, rx=-0.2145 ry=-3.1278 rz=-0.004 rad; joints [-48.359, -60.663, 91.816, -30.774, -229.681, 0.757] deg
                Waypoint Linea18_B: TCP in base x=-1150.106 y=624.337 z=110.084 mm, rx=1.1641 ry=-2.9058 rz=0.0105 rad; joints [-36.198, -18.752, 11.528, 7.722, -268.93, 0.895] deg
            Folder AB
              'desbaste_inicial'
              bajada_broca := p[0,0,-0.008,0,0,0]
              barrenos_menos1 := 19
              barreno_actual := 0
              Loop While (checkContinuously=false) expression=barreno_actual≤barrenos_menos1
                Folder Perforacion
                  MoveL speed 100 mm/s, acceleration 500 mm/s^2 (useActiveTCP=true) feature=Base
                    If barreno_actual≟6  or barreno_actual≟13
                      barreno_actual := barreno_actual+1
                    internos := interpolate_pose(Linea18_A, Linea18_B, barreno_actual/barrenos_menos1)
                    Waypoint Waypoint (Variable): variable=internos
                    'desbaste_inicial'
                    bajada_broca := p[0,0,-0.008,0,0,0]
                    bajada := p[0,0,0.008,0,0,0]
                    MoveDirectionNode (selectedDirection=ZMinus toolParams=0.003, 0.005)
                      Until DISTANCE (allowActions=false deceleration=3 distanceNodeType=STOP) Distance=0.045; motionParameters(blendRadius=0)
                    Popup Message (haltProgram=false message=punto contacto alanzdo inputType=Text)
                    MoveDirectionNode (selectedDirection=ZPlus toolParams=0.003, 0.005)
                      Until DISTANCE (allowActions=false deceleration=3 distanceNodeType=STOP) Distance=0.002; motionParameters(blendRadius=0)
                    Wait Sleep waitTime=0.3
                    Set DigitalOutput pin=config_out[1]; digitalValue=1
                    Wait Sleep waitTime=0.3
                    Loop Counting (count=3) loopVariable=Loop_133
                      bajar := pose_add(get_actual_tcp_pose(), bajada_broca)
                      Waypoint Waypoint (Variable): motionParameters(jointSpeed=1.047198 jointAcceleration=1.396263 cartesianSpeed=0.001 cartesianAcceleration=0.005); variable=bajar
                      subir := pose_sub(get_actual_tcp_pose(), bajada_broca)
                      Waypoint Waypoint (Variable): motionParameters(jointSpeed=1.047198 jointAcceleration=1.396263 cartesianSpeed=0.005 cartesianAcceleration=0.01); variable=subir
                      bajada_broca := pose_sub(bajada_broca, bajada)
                    MoveDirectionNode (selectedDirection=ZPlus toolParams=0.03, 0.035)
                      Until DISTANCE (allowActions=false deceleration=3 distanceNodeType=STOP) Distance=0.06; motionParameters(blendRadius=0)
                    Set DigitalOutput pin=config_out[1]; digitalValue=0
                    barreno_actual := barreno_actual+1
                    SuppressedNode
                      Call Quitar_broca
                    SuppressedNode
                      Call Poner_broca
          Popup Message (haltProgram=false message=Linea18 con chica Terminada! inputType=Text)
  'Subprogramas:'
SubProgram -> Quitar_broca
SubProgram -> Poner_broca
SubProgram Poner_broca (keepSynchronizedWithDisk=false)
  Folder Poner_broca
    If cambiar_broca≟ True  or iniciando_prog≟ True
      'Codigo de poner broca'
      Set DigitalOutput pin=ini_cambro_m289; digitalValue=0
      MoveL speed 250 mm/s, acceleration 1200 mm/s^2 (useActiveTCP=true) feature=Base
        If eje7≟2 and iniciando_prog≟ True
          Waypoint Home2: TCP in base x=-476.229 y=0 z=568.737 mm, rx=2.0263 ry=-2.3929 rz=-0.0208 rad; joints [-32.551, -116.469, 98.413, 17.843, -302.102, -0.163] deg
          Waypoint yendo1: TCP in base x=-246.137 y=407.69 z=568.737 mm, rx=-0.5894 ry=3.0844 rz=0.0228 rad; joints [-91.431, -116.469, 98.413, 17.843, -302.102, -0.163] deg
        If eje7≟3 and iniciando_prog≟ True
          Waypoint Home3: TCP in base x=-850.182 y=0 z=211.32 mm, rx=-2.0297 ry=2.3968 rz=0.0066 rad; joints [-14.374, -75.698, 98.757, -22.649, -284.037, -0.192] deg; TCP offset x=0.411 y=-218.298 z=37.994 mm, rx=1.558 ry=-0.1255 rz=0.1212 rad
          Waypoint Precam_bro1: TCP in base x=-795.771 y=128.511 z=757.632 mm, rx=1.5534 ry=-2.1987 rz=-0.8089 rad; joints [-24.356, -99.239, 84.164, -22.649, -284.037, -0.192] deg
          Waypoint Precam_bro2: TCP in base x=-204.472 y=779.716 z=757.632 mm, rx=-0.1114 ry=2.934 rz=1.0184 rad; joints [-90.488, -99.239, 84.164, -22.649, -284.037, -0.192] deg
        Waypoint Precambio_broca: TCP in base x=0.83 y=461.518 z=287.521 mm, rx=-0.2218 ry=-3.132 rz=0.0004 rad; joints [-125.124, -120.118, 128.54, -7.699, -306.118, -0.232] deg; TCP offset x=0.411 y=-218.298 z=37.994 mm, rx=1.558 ry=-0.1255 rz=0.1212 rad
        Popup Warning (haltProgram=false message=Cambia a las siguientes brocas inputType=Text)
        Waypoint Dejar_broca: motionParameters(jointSpeed=1.047198 jointAcceleration=1.396263 cartesianSpeed=0.09 cartesianAcceleration=0.1); TCP in base x=0.824 y=461.516 z=10.825 mm, rx=-0.2218 ry=-3.132 rz=0.0004 rad; joints [-125.105, -100.991, 150.063, -48.409, -306.183, -0.133] deg; TCP offset x=0.411 y=-218.298 z=37.994 mm, rx=1.558 ry=-0.1255 rz=0.1212 rad
      Set DigitalOutput pin=ini_cambro_m289; digitalValue=1
      Wait Sleep waitTime=2
      SuppressedNode
        Script: freedrive_mode()
      Wait Sleep waitTime=2
      Set DigitalOutput pin=ini_cambro_m289; digitalValue=0
      Wait Sleep waitTime=0.5
      Wait DigitalInput pin=fciclocarr_m292; digitalValue=0
      Wait Sleep waitTime=0.5
      SuppressedNode
        Script: end_freedrive_mode()
      MoveL speed 250 mm/s, acceleration 1200 mm/s^2 (useActiveTCP=true) feature=Base
        Waypoint Precambio_broca: motionParameters(jointSpeed=1.047198 jointAcceleration=1.396263 cartesianSpeed=0.09 cartesianAcceleration=0.1); TCP in base x=0.83 y=461.518 z=287.521 mm, rx=-0.2218 ry=-3.132 rz=0.0004 rad; joints [-125.124, -120.118, 128.54, -7.699, -306.118, -0.232] deg; TCP offset x=0.411 y=-218.298 z=37.994 mm, rx=1.558 ry=-0.1255 rz=0.1212 rad
        If eje7≟2
          Waypoint yendo1: TCP in base x=-246.137 y=407.69 z=568.737 mm, rx=-0.5894 ry=3.0844 rz=0.0228 rad; joints [-91.431, -116.469, 98.413, 17.843, -302.102, -0.163] deg
          Waypoint Home2: TCP in base x=-476.229 y=0 z=568.737 mm, rx=2.0263 ry=-2.3929 rz=-0.0208 rad; joints [-32.551, -116.469, 98.413, 17.843, -302.102, -0.163] deg
        If eje7≟3
          Waypoint Precam_bro2: TCP in base x=-204.472 y=779.716 z=757.632 mm, rx=-0.1114 ry=2.934 rz=1.0184 rad; joints [-90.488, -99.239, 84.164, -22.649, -284.037, -0.192] deg; TCP offset x=0.411 y=-218.298 z=37.994 mm, rx=1.558 ry=-0.1255 rz=0.1212 rad
          Waypoint Precam_bro1: TCP in base x=-795.771 y=128.511 z=757.632 mm, rx=1.5534 ry=-2.1987 rz=-0.8089 rad; joints [-24.356, -99.239, 84.164, -22.649, -284.037, -0.192] deg
          Waypoint Home3: TCP in base x=-850.182 y=0 z=211.32 mm, rx=-2.0297 ry=2.3968 rz=0.0066 rad; joints [-14.374, -75.698, 98.757, -22.649, -284.037, -0.192] deg
      barrenos_hechos := 0
      iniciando_prog := False
      cambiar_broca := False
    If barrenos_hechos≟14
      If cambiar_broca≟ False
        'Codigo de poner broca'
        Set DigitalOutput pin=ini_cambro_m289; digitalValue=0
        MoveL speed 250 mm/s, acceleration 1200 mm/s^2 (useActiveTCP=true) feature=Base
          Waypoint Precambio_broca: TCP in base x=0.83 y=461.518 z=287.521 mm, rx=-0.2218 ry=-3.132 rz=0.0004 rad; joints [-125.124, -120.118, 128.54, -7.699, -306.118, -0.232] deg; TCP offset x=0.411 y=-218.298 z=37.994 mm, rx=1.558 ry=-0.1255 rz=0.1212 rad
          Waypoint Dejar_broca: motionParameters(jointSpeed=1.047198 jointAcceleration=1.396263 cartesianSpeed=0.09 cartesianAcceleration=0.1); TCP in base x=0.824 y=461.516 z=10.825 mm, rx=-0.2218 ry=-3.132 rz=0.0004 rad; joints [-125.105, -100.991, 150.063, -48.409, -306.183, -0.133] deg; TCP offset x=0.411 y=-218.298 z=37.994 mm, rx=1.558 ry=-0.1255 rz=0.1212 rad
        Set DigitalOutput pin=ini_cambro_m289; digitalValue=1
        Wait Sleep waitTime=2
        SuppressedNode
          Script: freedrive_mode()
        Wait Sleep waitTime=2
        Set DigitalOutput pin=ini_cambro_m289; digitalValue=0
        Wait Sleep waitTime=0.5
        Wait DigitalInput pin=fciclocarr_m292; digitalValue=0
        Wait Sleep waitTime=0.5
        SuppressedNode
          Script: end_freedrive_mode()
        MoveL speed 250 mm/s, acceleration 1200 mm/s^2 (useActiveTCP=true) feature=Base
          Waypoint Precambio_broca: motionParameters(jointSpeed=1.047198 jointAcceleration=1.396263 cartesianSpeed=0.09 cartesianAcceleration=0.1); TCP in base x=0.83 y=461.518 z=287.521 mm, rx=-0.2218 ry=-3.132 rz=0.0004 rad; joints [-125.124, -120.118, 128.54, -7.699, -306.118, -0.232] deg; TCP offset x=0.411 y=-218.298 z=37.994 mm, rx=1.558 ry=-0.1255 rz=0.1212 rad
          If eje7≟2
            Waypoint yendo1: TCP in base x=-246.137 y=407.69 z=568.737 mm, rx=-0.5894 ry=3.0844 rz=0.0228 rad; joints [-91.431, -116.469, 98.413, 17.843, -302.102, -0.163] deg
            Waypoint Home2: TCP in base x=-476.229 y=0 z=568.737 mm, rx=2.0263 ry=-2.3929 rz=-0.0208 rad; joints [-32.551, -116.469, 98.413, 17.843, -302.102, -0.163] deg
          If eje7≟3
            Waypoint Precam_bro2: TCP in base x=-204.472 y=779.716 z=757.632 mm, rx=-0.1114 ry=2.934 rz=1.0184 rad; joints [-90.488, -99.239, 84.164, -22.649, -284.037, -0.192] deg; TCP offset x=0.411 y=-218.298 z=37.994 mm, rx=1.558 ry=-0.1255 rz=0.1212 rad
            Waypoint Precam_bro1: TCP in base x=-795.771 y=128.511 z=757.632 mm, rx=1.5534 ry=-2.1987 rz=-0.8089 rad; joints [-24.356, -99.239, 84.164, -22.649, -284.037, -0.192] deg
            Waypoint Home3: TCP in base x=-850.182 y=0 z=211.32 mm, rx=-2.0297 ry=2.3968 rz=0.0066 rad; joints [-14.374, -75.698, 98.757, -22.649, -284.037, -0.192] deg
        barrenos_hechos := 0
        iniciando_prog := False
        cambiar_broca := False
      Else 
        'Codigo de poner broca'
        Set DigitalOutput pin=ini_cambro_m289; digitalValue=0
        MoveL speed 250 mm/s, acceleration 1200 mm/s^2 (useActiveTCP=true) feature=Base
          Waypoint Precambio_broca: TCP in base x=0.83 y=461.518 z=287.521 mm, rx=-0.2218 ry=-3.132 rz=0.0004 rad; joints [-125.124, -120.118, 128.54, -7.699, -306.118, -0.232] deg; TCP offset x=0.411 y=-218.298 z=37.994 mm, rx=1.558 ry=-0.1255 rz=0.1212 rad
          Popup Warning (haltProgram=false message=Cambia a las siguientes brocas inputType=Text)
          Waypoint Dejar_broca: motionParameters(jointSpeed=1.047198 jointAcceleration=1.396263 cartesianSpeed=0.09 cartesianAcceleration=0.1); TCP in base x=0.824 y=461.516 z=10.825 mm, rx=-0.2218 ry=-3.132 rz=0.0004 rad; joints [-125.105, -100.991, 150.063, -48.409, -306.183, -0.133] deg; TCP offset x=0.411 y=-218.298 z=37.994 mm, rx=1.558 ry=-0.1255 rz=0.1212 rad
        Set DigitalOutput pin=ini_cambro_m289; digitalValue=1
        Wait Sleep waitTime=2
        SuppressedNode
          Script: freedrive_mode()
        Wait Sleep waitTime=2
        Set DigitalOutput pin=ini_cambro_m289; digitalValue=0
        Wait Sleep waitTime=0.5
        Wait DigitalInput pin=fciclocarr_m292; digitalValue=0
        Wait Sleep waitTime=0.5
        SuppressedNode
          Script: end_freedrive_mode()
        MoveL speed 250 mm/s, acceleration 1200 mm/s^2 (useActiveTCP=true) feature=Base
          Waypoint Precambio_broca: motionParameters(jointSpeed=1.047198 jointAcceleration=1.396263 cartesianSpeed=0.09 cartesianAcceleration=0.1); TCP in base x=0.83 y=461.518 z=287.521 mm, rx=-0.2218 ry=-3.132 rz=0.0004 rad; joints [-125.124, -120.118, 128.54, -7.699, -306.118, -0.232] deg; TCP offset x=0.411 y=-218.298 z=37.994 mm, rx=1.558 ry=-0.1255 rz=0.1212 rad
          If eje7≟2
            Waypoint yendo1: TCP in base x=-246.137 y=407.69 z=568.737 mm, rx=-0.5894 ry=3.0844 rz=0.0228 rad; joints [-91.431, -116.469, 98.413, 17.843, -302.102, -0.163] deg
            Waypoint Home2: TCP in base x=-476.229 y=0 z=568.737 mm, rx=2.0263 ry=-2.3929 rz=-0.0208 rad; joints [-32.551, -116.469, 98.413, 17.843, -302.102, -0.163] deg
          If eje7≟3
            Waypoint Precam_bro2: TCP in base x=-204.472 y=779.716 z=757.632 mm, rx=-0.1114 ry=2.934 rz=1.0184 rad; joints [-90.488, -99.239, 84.164, -22.649, -284.037, -0.192] deg; TCP offset x=0.411 y=-218.298 z=37.994 mm, rx=1.558 ry=-0.1255 rz=0.1212 rad
            Waypoint Precam_bro1: TCP in base x=-795.771 y=128.511 z=757.632 mm, rx=1.5534 ry=-2.1987 rz=-0.8089 rad; joints [-24.356, -99.239, 84.164, -22.649, -284.037, -0.192] deg
            Waypoint Home3: TCP in base x=-850.182 y=0 z=211.32 mm, rx=-2.0297 ry=2.3968 rz=0.0066 rad; joints [-14.374, -75.698, 98.757, -22.649, -284.037, -0.192] deg
        barrenos_hechos := 0
        iniciando_prog := False
        cambiar_broca := False
SubProgram Quitar_broca (keepSynchronizedWithDisk=false)
  Folder Quitar_broca
    barrenos_hechos := barrenos_hechos+1
    SuppressedNode
      Folder var
        SuppressedNode
          barrenos_hechos := 0
        eje7 := 2
        cambiar_broca := False
        iniciando_prog := False
    SuppressedNode
      ''
    If barrenos_hechos≟14 or cambiar_broca≟ True
      'Codigo de quitar broca'
      MoveL speed 250 mm/s, acceleration 1200 mm/s^2 (useActiveTCP=true) feature=Base
        MoveDirectionNode (selectedDirection=ZPlus)
          Until DISTANCE (allowActions=false deceleration=3 distanceNodeType=STOP) Distance=0.05; motionParameters(blendRadius=0)
        If eje7≟2
          Waypoint Home2: TCP in base x=-476.229 y=0 z=568.737 mm, rx=2.0263 ry=-2.3929 rz=-0.0208 rad; joints [-32.551, -116.469, 98.413, 17.843, -302.102, -0.163] deg; TCP offset x=0.411 y=-218.298 z=37.994 mm, rx=1.558 ry=-0.1255 rz=0.1212 rad
          Waypoint yendo1: TCP in base x=-246.137 y=407.69 z=568.737 mm, rx=-0.5894 ry=3.0844 rz=0.0228 rad; joints [-91.431, -116.469, 98.413, 17.843, -302.102, -0.163] deg
        If eje7≟3
          Waypoint Home3: TCP in base x=-850.182 y=0 z=211.32 mm, rx=-2.0297 ry=2.3968 rz=0.0066 rad; joints [-14.374, -75.698, 98.757, -22.649, -284.037, -0.192] deg; TCP offset x=0.411 y=-218.298 z=37.994 mm, rx=1.558 ry=-0.1255 rz=0.1212 rad
          Waypoint Precam_bro1: TCP in base x=-795.771 y=128.511 z=757.632 mm, rx=1.5534 ry=-2.1987 rz=-0.8089 rad; joints [-24.356, -99.239, 84.164, -22.649, -284.037, -0.192] deg
          Waypoint Precam_bro2: TCP in base x=-204.472 y=779.716 z=757.632 mm, rx=-0.1114 ry=2.934 rz=1.0184 rad; joints [-90.488, -99.239, 84.164, -22.649, -284.037, -0.192] deg
        Waypoint Precambio_broca: TCP in base x=0.83 y=461.518 z=287.521 mm, rx=-0.2218 ry=-3.132 rz=0.0004 rad; joints [-125.124, -120.118, 128.54, -7.699, -306.118, -0.232] deg; TCP offset x=0.411 y=-218.298 z=37.994 mm, rx=1.558 ry=-0.1255 rz=0.1212 rad
        Waypoint Dejar_broca: motionParameters(jointSpeed=1.047198 jointAcceleration=1.396263 cartesianSpeed=0.09 cartesianAcceleration=0.1); TCP in base x=0.824 y=461.516 z=10.825 mm, rx=-0.2218 ry=-3.132 rz=0.0004 rad; joints [-125.105, -100.991, 150.063, -48.409, -306.183, -0.133] deg; TCP offset x=0.411 y=-218.298 z=37.994 mm, rx=1.558 ry=-0.1255 rz=0.1212 rad
      Set DigitalOutput pin=outputbroc_m291; digitalValue=1
      Wait Sleep waitTime=2
      SuppressedNode
        Script: freedrive_mode()
      Wait Sleep waitTime=2
      Set DigitalOutput pin=outputbroc_m291; digitalValue=0
      Wait Sleep waitTime=0.5
      Wait DigitalInput pin=fciclocarr_m292; digitalValue=0
      Wait Sleep waitTime=0.5
      SuppressedNode
        Script: end_freedrive_mode()
      MoveL speed 250 mm/s, acceleration 1200 mm/s^2 (useActiveTCP=true) feature=Base
        Waypoint Precambio_broca: motionParameters(jointSpeed=1.047198 jointAcceleration=1.396263 cartesianSpeed=0.09 cartesianAcceleration=0.1); TCP in base x=0.83 y=461.518 z=287.521 mm, rx=-0.2218 ry=-3.132 rz=0.0004 rad; joints [-125.124, -120.118, 128.54, -7.699, -306.118, -0.232] deg; TCP offset x=0.411 y=-218.298 z=37.994 mm, rx=1.558 ry=-0.1255 rz=0.1212 rad
      Set DigitalOutput pin=avancarrusel_m7; digitalValue=1
      Wait Sleep waitTime=2
      Set DigitalOutput pin=avancarrusel_m7; digitalValue=0
      Wait Sleep waitTime=0.1
